INTERFACE ITF_TopElement1_HMI_Connector EXTENDS ITF_BaseTopElement_HMI_Connector,
	ITF_TopElement1_HMI_Connector_View, ITF_TopElement1_HMI_Connector_Command

END_INTERFACE

(* stored: Version 1.1.0.1
   Itf ITF_TopElement1_HMI_Connector: Id {bd8af3be-c60a-0222-0514-dafe7d1de7b9} *)
